// Alarm keypad interface
INTERFACE I_AlarmKeypad

// Returns true if the user input code equals the configured code
METHOD CheckCode : BOOL
END_METHOD

// Run this method every cycle
METHOD Execute
END_METHOD

// Returns the HMI data
PROPERTY HmiData : ST_AlarmKeypadHMI
GET
END_GET
END_PROPERTY

// Returns the keypad name
PROPERTY Name : STRING
GET
END_GET
END_PROPERTY

// Call this method once when the alarm state is changed
METHOD SetAlarmState
VAR_INPUT
	eAlarmState			: E_AlarmState;		// Alarm state
END_VAR
END_METHOD

// Set the buzzer command
METHOD SetBuzzer
VAR_INPUT
	eCommand	: E_DOCommand;
END_VAR
END_METHOD

// Set the keypad configured code
METHOD SetConfiguredCode
VAR_INPUT
	sCode	:	STRING;		// Configured code
END_VAR
END_METHOD

END_INTERFACE

(* stored: Version 1.1.0.1, ProductVersion 3.1.4024.12
   Itf I_AlarmKeypad: Id {e1af737e-7ada-48b3-84af-e4bed2430bb9}
   Folder Methods: Id {bd6d01f8-24c6-4c78-aad1-59ade80f0d13}
   Folder Properties: Id {9df19c54-276b-408b-a285-4a5c9406e214}
   Method CheckCode: Id {2124e254-5d12-4552-937d-aaf5ddbb14e5}
   Method Execute: Id {6687a198-5bd5-408e-bb2d-a604220d5d1b}
   Property HmiData: Id {0899eb50-bd5e-49fb-8c99-2af9f87ea4ea}
   Get Get: Id {c683d460-093d-49fe-98b1-cb646f988449}
   Property Name: Id {09c3cce0-5fb9-489a-9d79-9510a910ca81}
   Get Get: Id {43954b39-90aa-4dbc-9a73-724a16de966d}
   Method SetAlarmState: Id {1b0a1209-7f0d-485f-bb60-2c6ea6f8cf32}
   Method SetBuzzer: Id {f79373aa-4fb1-449f-a534-4040e85e3a7f}
   Method SetConfiguredCode: Id {ff808e38-20da-40e3-8366-da25a37d4048} *)
